INTERFACE Alarm

METHOD Clear
VAR_INPUT
END_VAR
END_METHOD

METHOD ClearArguments : I_TcArguments
END_METHOD

{attribute 'monitoring' := 'call'}
PROPERTY IsRaised : BOOL
GET
END_GET
END_PROPERTY

METHOD Raise
VAR_INPUT
END_VAR
END_METHOD

{attribute 'monitoring' := 'call'}
PROPERTY Source : Name
GET
END_GET
SET
END_SET
END_PROPERTY

END_INTERFACE

(* stored: Version 1.1.0.1
   Itf Alarm: Id {a115ae59-9c39-0ffc-3485-220b1d762515}
   Method Clear: Id {6a5e9cf1-e645-0394-369e-44b9089f83a3}
   Method ClearArguments: Id {fb0c6a84-23e5-0d10-2cb4-47a090e3622a}
   Property IsRaised: Id {4098fd7e-9c07-0d75-201d-740ac9de4e6b}
   Get Get: Id {a5c5cae1-e0db-0406-1a41-15792b100a52}
   Method Raise: Id {bd03e23d-0bd6-0593-2919-8f55a4b6e34c}
   Property Source: Id {89716997-9da2-0867-13e3-3b1ee50ea82d}
   Get Get: Id {82446f50-cc19-008c-2847-ab3ac2c7b4ba}
   Set Set: Id {eec35149-2350-0873-2647-ad4c4025d295} *)
